FUNCTION_BLOCK FB_HandshakeDelay	// Delays the signal (TOF) so the handshake has enough time to be seen by the other part (inside PLC/EAP/normal IO)
VAR_INPUT
	iHandshake:			BOOL;				// The handshake signal
	iSignalDuration:	TIME := T#100MS;	// The delay
END_VAR
VAR_OUTPUT
	oHandshake:	BOOL;						// The handshake signal having an additional delay
END_VAR
VAR
	delay: TOF;
END_VAR

delay(IN := iHandshake, PT := iSignalDuration, Q => oHandshake);

END_FUNCTION_BLOCK

(* stored: Version 1.1.0.1, ProductVersion 3.1.4026.18
   POU FB_HandshakeDelay: Id {30d03d4e-0a9e-4968-a5a5-65b67a51fb54}, SpecialFunc None *)
